Staubli VAL3: deleteAll.pgx

public program deleteAll(num x_nType)
  local num i
  local num nSize[3]
begin
  // onEvent
  call OnEvent:OnCycleEvent(15)
  //
  logMsg("[KERNEL] CYCLE:Delete all the program..")
  call getSize(nSize,x_nType)
  for i=0 to (nSize-1)
    call delete(0,x_nType)
  endFor
  // reinit the buffer of all the program
  // cycleStatus:bInitMemory=true
end
